// TIA Portal V19 export
DATA_BLOCK "A0301_Fermi_P4"   // DB46
// stored: InstanceOfName A0301_Fermi_P4_FB, InstanceOfType FB
"A0301_Fermi_P4_FB"
   // VAR_INPUT
   //    AreaInterface : "AreaInterface";
   //    ZSI : "udt_ZoneSafetyInterface";
   //    DSI : "udt_DeviceSafetyInterface";
   //    DataIn : Struct
   //       OP_Rest_PB : Bool;
   //       OP_Work_PB : Bool;
   //    END_STRUCT;
   //    CIn : Struct
   //       Manager : "ValveMachine_Manager";
   //       SemiAut_Pb : Bool;
   //       P3 : Struct
   //          Fermi : "ValveMachine_COut";
   //       END_STRUCT;
   //       Trasporto : "SpeedMachine_COut";
   //    END_STRUCT;
   //    Config : Struct
   //       Fermi : Array[1..6] of "ValveMachine_Config";
   //       DelayMissingCondition : Time;
   //    END_STRUCT;
   // END_VAR
   // VAR_OUTPUT
   //    MachineInterface : "MachineInterface";
   //    COut : Struct
   //       Fermi : "ValveMachine_COut";
   //    END_STRUCT;
   // END_VAR
   // VAR
   //    Alarm : Struct
   //       Fermi : Array[1..6] of "ValveAlr";
   //    END_STRUCT;
   //    Warning : Struct
   //       Fermi : Array[1..6] of "ValveMachine_Wng";
   //       OP_REST_MissingCnd : Bool;
   //       OP_WORK_MissingCnd : Bool;
   //    END_STRUCT;
   //    HMI : Struct
   //       Selection : Array[1..6] of Bool;
   //       FermiSts { S7_SetPoint := 'True'} : "UDT_HMI-Sts_ValvePosA0301";
   //    END_STRUCT;
   //    Sts : Struct
   //       Fermi_AlarmPresence : Bool;
   //       OP_CanMoveFreely : Bool;
   //       OP_Rest_Cnd : Bool;
   //       Op_Work_Cnd : Bool;
   //    END_STRUCT;
   //    Ctrl : Struct
   //       OP_Rest_Man : Bool;
   //       OP_Work_Man : Bool;
   //       OP_Rest_Aut : Bool;
   //       OP_Work_Aut : Bool;
   //       OP_Rest : Bool;
   //       OP_Work : Bool;
   //    END_STRUCT;
   //    Fermi { S7_SetPoint := 'True'} : Array[1..6] of "ValveMachine_FB";
   //    AUX : Struct
   //       OP_Rest_PB : Bool;
   //       OP_Work_PB : Bool;
   //    END_STRUCT;
   //    TON_OP_REST_MissingCnd { S7_SetPoint := 'True'} : TON_TIME;
   //    TON_OP_WORK_MissingCnd { S7_SetPoint := 'True'} : TON_TIME;
   // END_VAR
BEGIN
   HMI.Selection[1..6] := TRUE;
END_DATA_BLOCK
